# B&R Automation Studio project PLC_base3
Automation Studio 

## Logical view

### Global.var
```iecst
VAR
	data1 : STRING[1000];
	data2 : STRING[1000];
	activeData : USINT;
	readyForData : BOOL;
	receivedData : BOOL;
	readyToConvert : BOOL;
	instSize : DINT;
	instructionsArray : ARRAY[0..999] OF STRING[25];
	xArray : ARRAY[0..100] OF INT;
	yArray : ARRAY[0..100] OF INT;
	zArray : ARRAY[0..100] OF INT;
END_VAR
```

### Program Logical/Program

#### Types.typ
```iecst
TYPE
	ROBOSTATE2 :
		(
		INIT,
		READY,
		RECEIVE,
		CONVERT,
		RESET,
		CALIBRATE,
		MANUAL,
		DRAW,
		DRAW2,
		BACK,
		NEXTLINE,
		PENCILDOWN,
		PENCILUP,
		SHARPEN,
		STOP
		);
END_TYPE
```

#### Variables.var
```iecst
(*CONVERSION*)
VAR
	yPrev : INT;
	counter : UINT;
	delim1 : STRING[80];
	delim2 : STRING[80];
	string1 : STRING[80];
	string2 : STRING[80];
	D1 : INT;
	D2 : INT;
	D3 : INT;
	D4 : INT;
	D5 : INT;
	D6 : INT;
	x1 : INT;
	y1 : INT;
	x2 : INT;
	y2 : INT;
	z1 : INT;
	z2 : INT;
END_VAR
(*MOVEMENT*)
VAR
	ROBOSTATE : ROBOSTATE2;
	xCalib : DINT;
	yCalib : DINT;
	zCalib : DINT;
	count : DINT;
	sharpener : {REDUND_UNREPLICABLE} BOOL;
	xEnable : {REDUND_UNREPLICABLE} BOOL;
	yEnable : {REDUND_UNREPLICABLE} BOOL;
	zEnable : {REDUND_UNREPLICABLE} BOOL;
	StopMaskine : BOOL;
	Programsteps : UINT;
	xCounter : DINT;
	yCounter : DINT;
	zCounter : DINT;
	xDirection : BOOL;
	yDirection : BOOL;
	zDirection : BOOL;
	xNext : BOOL;
	yNext : BOOL;
	zNext : BOOL;
	xStep : BOOL;
	yStep : BOOL;
	zStep : BOOL;
	xNegMove : BOOL;
	yNegMove : BOOL;
	zNegMove : BOOL;
	xPosMove : BOOL;
	yPosMove : BOOL;
	zPosMove : BOOL;
	bStop : BOOL;
	xStop : BOOL;
	yStop : BOOL;
	zStop : BOOL;
	scale : DINT;
	start1 : BOOL;
	timer : TON;
	killswitch : BOOL;
	hasBeenSharpened : BOOL;
END_VAR
```

#### Main.st
```iecst
PROGRAM _INIT
	ROBOSTATE := READY;

	counter := 0;
	delim1 := ' ';
	delim2 := ',';

	xEnable := FALSE;
	yEnable := FALSE;
	zEnable := FALSE;

	count := 0;
	xCounter := 0;
	yCounter := 0;
	zCounter := 0;
	xCalib := 0; //17680
	yCalib := 0; //13364
	zCalib := 0;
	yPrev := 0;
	xNext := FALSE;
	yNext := FALSE;
	zNext := FALSE;
	xDirection := FALSE;
	yDirection := FALSE;
	zDirection := FALSE;
	xStep := FALSE;
	yStep := FALSE;
	zStep := FALSE;
	xNegMove := FALSE;
	yNegMove := FALSE;
	zNegMove := FALSE;
	xPosMove := FALSE;
	yPosMove := FALSE;
	zPosMove := FALSE;
	hasBeenSharpened := TRUE;
	scale := 25; // steps / px
END_PROGRAM

PROGRAM _CYCLIC
	IF killswitch THEN // Killswitch to stop robot in case of emergency
		//ROBOSTATE := STOP;
	END_IF;

	CASE ROBOSTATE OF
		INIT:
			counter := 0;
			delim1 := ' ';
			delim2 := ',';

			xEnable := FALSE;
			yEnable := FALSE;
			zEnable := FALSE;

			count := 0;
			xCounter := 0;
			yCounter := 0;
			zCounter := 0;
			xCalib := 0; //17680
			yCalib := 0; //13364
			zCalib := 0;
			yPrev := 0;
			xNext := FALSE;
			yNext := FALSE;
			zNext := FALSE;
			xDirection := FALSE;
			yDirection := FALSE;
			zDirection := FALSE;
			xStep := FALSE;
			yStep := FALSE;
			zStep := FALSE;
			xNegMove := FALSE;
			yNegMove := FALSE;
			zNegMove := FALSE;
			xPosMove := FALSE;
			yPosMove := FALSE;
			zPosMove := FALSE;
			readyToConvert := FALSE;
			scale := 25;

			FOR count := 0 TO 999 DO
				instructionsArray[count] := '';
				xArray[count] := 0;
				yArray[count] := 0;
				zArray[count] := 0;
			END_FOR;

			ROBOSTATE := READY;

		READY: // Does nothing, is meant to wait until finished receiving instructions
			IF (readyToConvert = TRUE) THEN
				ROBOSTATE := CONVERT;
			END_IF

		CONVERT:
			timer(IN := NOT timer.Q, PT := T#100ms);
			IF (timer.Q = TRUE) THEN
				IF (counter < (instSize)) THEN
					// Splits element on index counter of instructionsArray[] into two seperate strings
					string1 := LEFT(instructionsArray[counter], FIND(instructionsArray[counter], delim2));
					string2 := RIGHT(instructionsArray[counter], FIND(instructionsArray[counter], delim2));

					// Finds numerical positions of all delimiters " " and "," in both strings
					D1 := FIND(string1, delim1);
					D2 := FIND(string1, delim1) + D1;
					D3 := FIND(string1, delim2);
					D4 := FIND(string2, delim1);
					D5 := FIND(string2, delim1) + D4;
					D6 := FIND(string2, delim2);

					// Isolates coordinates into individual integers
					xArray[counter] := STRING_TO_INT(LEFT(string1, D1 - 1));
					yArray[counter] := STRING_TO_INT(MID(string1, D2 - D1 - 1, D1 + 1));
					zArray[counter] := STRING_TO_INT(MID(string1, D3 - D2 - 1, D2 + 1));

					xArray[counter + 1] := STRING_TO_INT(LEFT(string2, D4 - 1));
					yArray[counter + 1] := STRING_TO_INT(MID(string2, D5 - D4 - 1, D4 + 1));
					zArray[counter + 1] := STRING_TO_INT(MID(string2, D6 - D5 - 1, D5 + 1));
					counter := counter + 2;
				ELSE
					ROBOSTATE := RESET;

					counter := 0;
				END_IF
			END_IF

		MANUAL:
			IF (killswitch <> TRUE) THEN
				IF (xStop <> TRUE OR xCounter > 0) THEN
					IF (xPosMove = TRUE) THEN
						IF (xPosMove = xNegMove) THEN
							xPosMove := FALSE;
						END_IF
						xDirection := TRUE;
						xStep := NOT xStep;
						xCounter := xCounter + 1;
					END_IF

					IF (xNegMove = TRUE) THEN
						IF (xPosMove = xNegMove) THEN
							xNegMove := FALSE;
						END_IF
						xDirection := FALSE;
						xStep := NOT xStep;
						xCounter := xCounter - 1;
					END_IF
				END_IF

				IF (yStop <> TRUE OR yCounter > 0) THEN
					IF (yPosMove = TRUE) THEN
						IF (yPosMove = yNegMove) THEN
							yPosMove := FALSE;
						END_IF
						yDirection := TRUE;
						yStep := NOT yStep;
						yCounter := yCounter + 1;
					END_IF

					IF (yNegMove = TRUE) THEN
						IF (yPosMove = yNegMove) THEN
							yNegMove := FALSE;
						END_IF
						yDirection := FALSE;
						yStep := NOT yStep;
						yCounter := yCounter - 1;
					END_IF
				END_IF

				IF (zCounter >= 0 AND zCounter <= 7500) THEN
					IF (zPosMove = TRUE) THEN
						IF (zPosMove = zNegMove) THEN
							zPosMove := FALSE;
						END_IF
						zDirection := TRUE;
						zStep := NOT zStep;
						zCounter := zCounter - 1;
					END_IF

					IF (zNegMove = TRUE) THEN
						IF (zPosMove = zNegMove) THEN
							zNegMove := FALSE;
						END_IF
						zDirection := FALSE;
						zStep := NOT zStep;
						zCounter := zCounter + 1;
					END_IF
				END_IF
			END_IF

		DRAW:
			IF (killswitch <> TRUE OR counter < instSize) THEN
				IF (xStop <> TRUE) THEN
					IF (xArray[counter] * scale > xCounter) THEN
						xNext := FALSE;
						xDirection := TRUE;
						xStep := NOT xStep;
						xCounter := xCounter + 1;
					ELSIF (xArray[counter] * scale < xCounter) THEN
						xNext := FALSE;
						xDirection := FALSE;
						xStep := NOT xStep;
						xCounter := xCounter - 1;
					ELSIF (xArray[counter] * scale = xCounter AND xNext = FALSE) THEN
						ROBOSTATE := PENCILDOWN;
					END_IF
				END_IF
			END_IF

		DRAW2:
			IF (killswitch <> TRUE) THEN
				IF (xStop <> TRUE) THEN
					IF (xArray[counter + 1] * scale > xCounter) THEN
						xNext := FALSE;
						xDirection := TRUE;
						xStep := NOT xStep;
						xCounter := xCounter + 1;
					ELSIF (xArray[counter + 1] * scale < xCounter) THEN
						xNext := FALSE;
						xDirection := FALSE;
						xStep := NOT xStep;
						xCounter := xCounter - 1;
					ELSIF (xArray[counter + 1] * scale = xCounter AND xNext = FALSE) THEN
						ROBOSTATE := PENCILUP;
					END_IF
				END_IF
			END_IF

		NEXTLINE:
			IF (killswitch <> TRUE) THEN
				IF (yStop <> TRUE) THEN
					IF (yArray[counter + 1] <> yArray[counter] AND (counter MOD(50)) <> 0 AND hasBeenSharpened = TRUE) THEN
						yDirection := TRUE;
						yStep := NOT yStep;
						yCounter := yCounter + 1;
					ELSIF (yArray[counter + 1] = yArray[counter]) THEN
						ROBOSTATE := DRAW;
					ELSIF ((counter MOD(50)) = 0 AND hasBeenSharpened = TRUE) THEN
						hasBeenSharpened := FALSE;
						ROBOSTATE := SHARPEN;
					END_IF
				END_IF
			END_IF

		PENCILDOWN:
			IF (killswitch <> TRUE) THEN
				IF (bStop <> TRUE) THEN
					zDirection := TRUE;
					zStep := NOT zStep;
					zCounter := zCounter - 1;
				ELSE
					ROBOSTATE := DRAW2;
				END_IF
			END_IF
		PENCILUP:
			IF (killswitch <> TRUE) THEN
				IF (zCounter < 500) THEN
					zDirection := FALSE;
					zStep := NOT zStep;
					zCounter := zCounter + 1;
				ELSE
					counter := counter + 1;
					ROBOSTATE := NEXTLINE;
				END_IF
			END_IF

		SHARPEN:
			IF (killswitch <> TRUE) THEN
				IF (zCounter < 3500 AND zStop <> TRUE AND xStop <> TRUE) THEN
					zDirection := FALSE;
					zStep := NOT zStep;
					zCounter := zCounter + 1;
				ELSIF (zCounter >= 3500 AND xStop <> TRUE AND zStop <> TRUE) THEN
					xDirection := FALSE;
					xStep := NOT xStep;
					xCounter := xCounter - 1;
				ELSIF (xStop = TRUE AND zStop <> TRUE) THEN
					IF (hasBeenSharpened <> TRUE AND zCounter > 1450) THEN
						sharpener := TRUE;
						zDirection := TRUE;
						zStep := NOT zStep;
						zCounter := zCounter - 1;
					ELSIF (zCounter = 1450) THEN
						timer(IN := NOT timer.Q, PT := T#2500ms);
						hasBeenSharpened := TRUE;
					END_IF
					IF (zCounter < 3500 AND hasBeenSharpened = TRUE AND timer.Q) THEN
						sharpener := FALSE;
						zDirection := FALSE;
						zStep := NOT zStep;
						zCounter := zCounter + 1;
					ELSIF (zCounter >= 3500 AND hasBeenSharpened = TRUE) THEN
						ROBOSTATE := BACK;
					END_IF
				END_IF
			END_IF

		BACK:
			IF (killswitch <> TRUE) THEN
				IF (xArray[counter] * scale > xCounter AND hasBeenSharpened = TRUE) THEN
					xDirection := TRUE;
					xStep := NOT xStep;
					xCounter := xCounter + 1;
				ELSIF (xArray[counter] * scale = xCounter AND bStop <> TRUE AND hasBeenSharpened = TRUE) THEN
					zDirection := TRUE;
					zStep := NOT zStep;
					zCounter := zCounter - 1;
				ELSIF (xArray[counter] * scale = xCounter AND bStop = TRUE AND hasBeenSharpened = TRUE) THEN
					ROBOSTATE := DRAW;
				END_IF
			END_IF

		RESET: // ASSUMES XCALIB AND YCALIB AS CONTAINING MAX STEPS ON X AND Y AXIS AS IT USES THESE TO FIND ORIGO
			sharpener := FALSE;
			IF (killswitch <> TRUE) THEN
				zCalib := 0;
				IF (zStop <> TRUE) THEN
					zDirection := FALSE;
					zStep := NOT zStep;
					zCounter := zCounter + 1;
				ELSE
					zCounter := zCalib;
				END_IF
				IF (xStop <> TRUE AND zStop = TRUE) THEN
					xDirection := FALSE;
					xStep := NOT xStep;
					xCounter := xCounter + 1;
				ELSE
					xCounter := xCalib;
				END_IF
				IF (yStop <> TRUE AND zStop = TRUE) THEN
					yDirection := FALSE;
					yStep := NOT yStep;
					yCounter := yCounter + 1;
				ELSE
					yCounter := yCalib;
				END_IF

				IF (xStop = TRUE AND yStop = TRUE AND zStop = TRUE) THEN
					ROBOSTATE := CALIBRATE;
				END_IF
			END_IF

		CALIBRATE: // ONLY USE CALIBRATE IF ALL STOP SENSORS ARE ACTIVATED
			IF (xCounter < 3280) THEN
				xDirection := TRUE;
				xStep := NOT xStep;
				xCounter := xCounter + 1;
			END_IF
			IF (yCounter < 1364) THEN
				yDirection := TRUE;
				yStep := NOT yStep;
				yCounter := yCounter + 1;
			END_IF
			IF (xCounter >= 3280 AND xCounter <= 17680 AND yCounter >= 1364 AND yCounter <= 13364) THEN
				IF (bStop <> TRUE AND zPosMove = FALSE) THEN
					zDirection := TRUE;
					zStep := NOT zStep;
					zCounter := zCounter + 1;
				ELSIF (bStop = TRUE AND zPosMove = FALSE) THEN
					zPosMove := TRUE;
					zCounter := 0;
				ELSIF (zPosMove = TRUE) THEN
					IF (zCounter < 500) THEN
						zDirection := FALSE;
						zStep := NOT zStep;
						zCounter := zCounter + 1;
					ELSE
						zPosMove := FALSE;
						xCounter := 0;
						yCounter := 0;
						ROBOSTATE := MANUAL;
					END_IF
				END_IF
			END_IF
	END_CASE
END_PROGRAM

PROGRAM _EXIT

END_PROGRAM
```

### Program Logical/Socket

#### Types.typ
```iecst
TYPE
	TCPSTATE :
		(
		TCPSTATE_CLOSE,
		TCPSTATE_SEND,
		TCPSTATE_RECEIVE,
		TCPSTATE_SERVER_CREATE,
		TCPSTATE_SOCKET_OPEN,
		TCPSTATE_RESET
	);
END_TYPE
```

#### Variables.var
```iecst
VAR
	receiveData : STRING[80];
	sendData : STRING[80];
	TcpClose1 : TcpClose;
	TcpClose2 : TcpClose;
	TcpOpen1 : TcpOpen;
	TcpReceive1 : TcpRecv;
	TcpSend1 : TcpSend;
	TcpServer1 : TcpServer;
	tcpst : TCPSTATE;
	testUA : INT;
	timer : TON;
	firstData : BOOL;
	moreData : BOOL;
	count : DINT;
END_VAR
```

#### Main.st
```iecst
PROGRAM _INIT
	tcpst := TCPSTATE_SOCKET_OPEN;

	data1 := '';
	data2 := '';
	activeData := 2;
	readyForData := TRUE;
	firstData := TRUE;
	receivedData := FALSE;
	moreData := FALSE;
	receiveData := '';
	FOR count := 0 TO 999 DO
		instructionsArray[count] := '';
		xArray[count] := 0;
		yArray[count] := 0;
		zArray[count] := 0;
	END_FOR;
	count := 0;
	readyToConvert := FALSE;
END_PROGRAM

PROGRAM _CYCLIC
	CASE tcpst OF
		TCPSTATE_SOCKET_OPEN: // Open socket for connection
			TcpOpen1.enable := TRUE;
			TcpOpen1.port := 12345;
			TcpOpen1.options := tcpOPT_REUSEADDR;
			TcpOpen1();
			IF (TcpOpen1.status = ERR_OK) THEN
				tcpst := TCPSTATE_SERVER_CREATE;
			END_IF

		TCPSTATE_SERVER_CREATE: // Connect to Java side
			TcpServer1.enable := TRUE;
			TcpServer1.ident := TcpOpen1.ident;
			TcpServer1();
			IF (TcpServer1.status = ERR_OK) THEN
				tcpst := TCPSTATE_RECEIVE;
			END_IF

		TCPSTATE_RECEIVE: // Prepare to receive data
			IF (readyForData) THEN
				TcpReceive1.enable := TRUE;
				TcpReceive1.ident := TcpServer1.identclnt;
				TcpReceive1.pData := ADR(receiveData);
				TcpReceive1.datamax := SIZEOF(receiveData);
				TcpReceive1();
				IF (TcpReceive1.status = ERR_OK) THEN
					tcpst := TCPSTATE_RECEIVE;
					// Select right data buffer and store coordinates in instructionsArray[]
					IF (activeData = 1) THEN
						data2 := '';
						data2 := LEFT(receiveData, UDINT_TO_INT(TcpReceive1.recvlen));
						IF (data2 <> 'DONE') THEN
							instructionsArray[count] := data2;
						ELSE
							instSize := count;
							readyToConvert := TRUE;
						END_IF
					ELSE
						data1 := '';
						data1 := LEFT(receiveData, UDINT_TO_INT(TcpReceive1.recvlen));
						IF (data1 <> 'DONE') THEN
							instructionsArray[count] := data1;
						ELSE
							instSize := count;
							readyToConvert := TRUE;
						END_IF

					END_IF

					// Important: set variables that is changed by higher priority tasks
					// before the control variable
					readyForData := FALSE;
					receivedData := TRUE;
					count := count + 1;
				END_IF
			END_IF
			IF (TcpSend1.status = ERR_OK) THEN
				tcpst := TCPSTATE_RECEIVE;
			END_IF

		TCPSTATE_SEND: // Send OK back to Java side, to signal successful receiving of data
			sendData := 'OK';
			TcpSend1.enable := TRUE;
			TcpSend1.ident := TcpServer1.identclnt;
			TcpSend1.pData := ADR(sendData);
			TcpSend1.datalen := brsstrlen(ADR(sendData)); // Uses brsstrlen() to get the length in UDINT datatype
			TcpSend1();
			IF (TcpSend1.status = ERR_OK) THEN
				tcpst := TCPSTATE_RECEIVE;
			END_IF

		TCPSTATE_CLOSE: // Close TCP socket and reset data variables
			TcpClose1.enable := TRUE;
			TcpClose1.ident := TcpServer1.identclnt;
			TcpClose1();

			data1 := '';
			data2 := '';
			activeData := 2;
			readyForData := TRUE;
			firstData := TRUE;
			receivedData := FALSE;
			moreData := FALSE;
			receiveData := '';
			FOR count := 0 TO 249 DO
				instructionsArray[count] := '';
			END_FOR;
			count := 0;

			IF (TcpClose1.status = ERR_OK) THEN
				TcpServer1.enable := FALSE;
				TcpServer1();
				tcpst := TCPSTATE_SERVER_CREATE;
			END_IF

		TCPSTATE_RESET:	// Reset data variables
			data1 := '';
			data2 := '';
			activeData := 2;
			readyForData := TRUE;
			firstData := TRUE;
			receivedData := FALSE;
			moreData := FALSE;
			receiveData := '';
			FOR count := 0 TO 999 DO
				instructionsArray[count] := '';
				xArray[count] := 0;
				yArray[count] := 0;
				zArray[count] := 0;
			END_FOR;
			count := 0;
			tcpst := TCPSTATE_RECEIVE;
	END_CASE

	// Double buffer part of code
	timer(IN := NOT timer.Q, PT := T#100ms);

	IF (receivedData) THEN
		readyForData := FALSE;
		receivedData := FALSE;
		moreData := TRUE;

		IF (firstData) THEN
			firstData := FALSE;
			readyForData := TRUE;
			IF (activeData = 2) THEN
				activeData := 1;
			ELSE
				activeData := 2;
			END_IF
		END_IF;
	END_IF;

	IF (timer.Q) THEN
		IF (moreData) THEN
			moreData := FALSE;

			IF (activeData = 2) THEN
				activeData := 1;
			ELSE
				activeData := 2;
			END_IF
		ELSE
			firstData := TRUE;
		END_IF
		readyForData := TRUE;
	END_IF

END_PROGRAM

PROGRAM _EXIT
	TcpClose1.enable := TRUE;
	TcpClose1.ident := TcpServer1.identclnt;
	TcpClose1();

	TcpClose2.enable := TRUE;
	TcpClose2.ident := TcpOpen1.ident;
	TcpClose2();
END_PROGRAM
```
